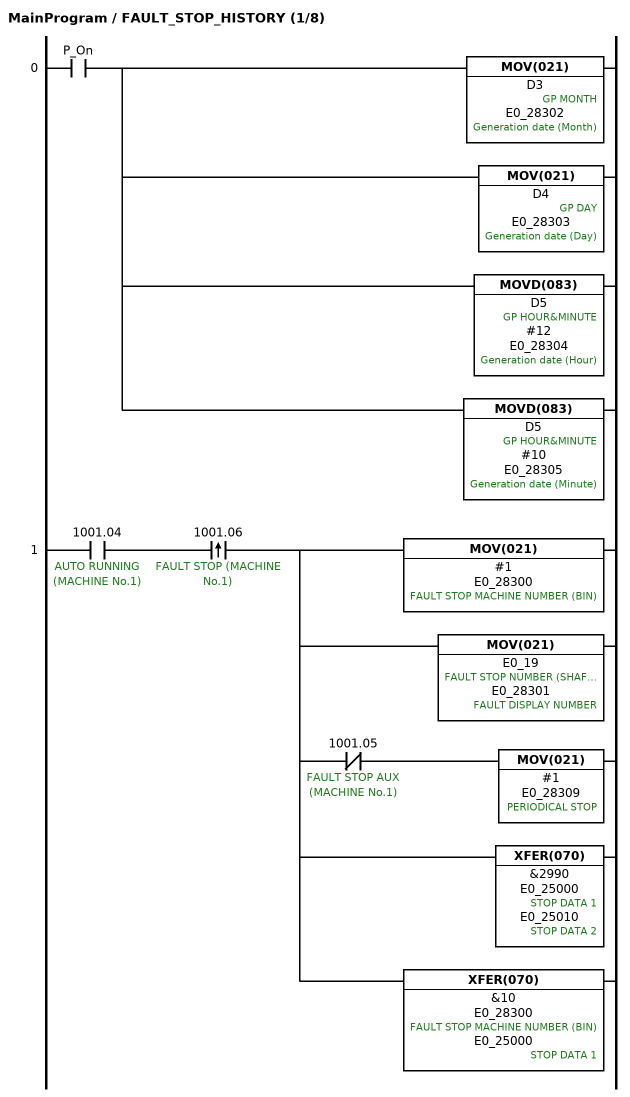
; [picture p168: MainProgram / FAULT_STOP_HISTORY, rungs 0-1]
; rung 0
LD P_On
MOV(021) D3 E0_28302  ; GP MONTH, Generation date (Month)
MOV(021) D4 E0_28303  ; GP DAY, Generation date (Day)
MOVD(083) D5 #12 E0_28304  ; GP HOUR&MINUTE, Generation date (Hour)
MOVD(083) D5 #10 E0_28305  ; GP HOUR&MINUTE, Generation date (Minute)
; rung 1
LD 1001.04  ; AUTO RUNNING (MACHINE No.1)
@AND 1001.06  ; FAULT STOP (MACHINE No.1)
OUT TR0
MOV(021) #1 E0_28300  ; FAULT STOP MACHINE NUMBER (BIN)
MOV(021) E0_19 E0_28301  ; FAULT STOP NUMBER (SHAFT PRESS-FITTING), FAULT DISPLAY NUMBER
ANDNOT 1001.05  ; FAULT STOP AUX (MACHINE No.1)
MOV(021) #1 E0_28309  ; PERIODICAL STOP
LD TR0
XFER(070) &2990 E0_25000 E0_25010  ; STOP DATA 1, STOP DATA 2
XFER(070) &10 E0_28300 E0_25000  ; FAULT STOP MACHINE NUMBER (BIN), STOP DATA 1

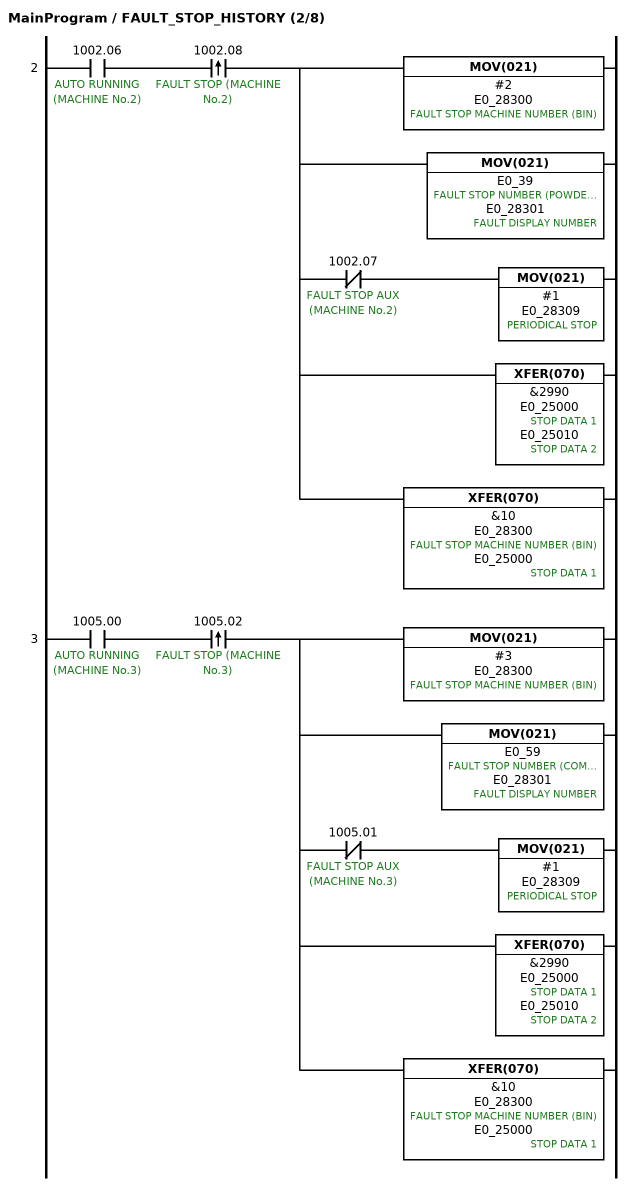
; rung 2
LD 1002.06  ; AUTO RUNNING (MACHINE No.2)
@AND 1002.08  ; FAULT STOP (MACHINE No.2)
OUT TR0
MOV(021) #2 E0_28300  ; FAULT STOP MACHINE NUMBER (BIN)
MOV(021) E0_39 E0_28301  ; FAULT STOP NUMBER (POWDER COATING), FAULT DISPLAY NUMBER
ANDNOT 1002.07  ; FAULT STOP AUX (MACHINE No.2)
MOV(021) #1 E0_28309  ; PERIODICAL STOP
LD TR0
XFER(070) &2990 E0_25000 E0_25010  ; STOP DATA 1, STOP DATA 2
XFER(070) &10 E0_28300 E0_25000  ; FAULT STOP MACHINE NUMBER (BIN), STOP DATA 1
; rung 3
LD 1005.00  ; AUTO RUNNING (MACHINE No.3)
@AND 1005.02  ; FAULT STOP (MACHINE No.3)
OUT TR0
MOV(021) #3 E0_28300  ; FAULT STOP MACHINE NUMBER (BIN)
MOV(021) E0_59 E0_28301  ; FAULT STOP NUMBER (COMM PRESS-FITTING), FAULT DISPLAY NUMBER
ANDNOT 1005.01  ; FAULT STOP AUX (MACHINE No.3)
MOV(021) #1 E0_28309  ; PERIODICAL STOP
LD TR0
XFER(070) &2990 E0_25000 E0_25010  ; STOP DATA 1, STOP DATA 2
XFER(070) &10 E0_28300 E0_25000  ; FAULT STOP MACHINE NUMBER (BIN), STOP DATA 1

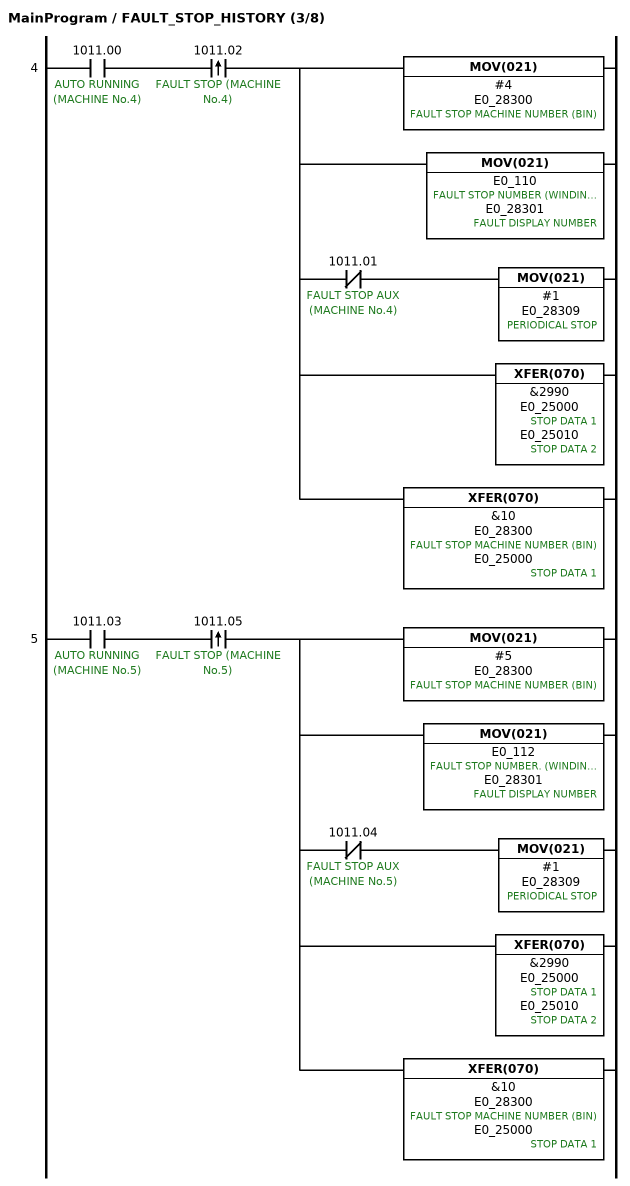
; rung 4
LD 1011.00  ; AUTO RUNNING (MACHINE No.4)
@AND 1011.02  ; FAULT STOP (MACHINE No.4)
OUT TR0
MOV(021) #4 E0_28300  ; FAULT STOP MACHINE NUMBER (BIN)
MOV(021) E0_110 E0_28301  ; FAULT STOP NUMBER (WINDING No.1), FAULT DISPLAY NUMBER
ANDNOT 1011.01  ; FAULT STOP AUX (MACHINE No.4)
MOV(021) #1 E0_28309  ; PERIODICAL STOP
LD TR0
XFER(070) &2990 E0_25000 E0_25010  ; STOP DATA 1, STOP DATA 2
XFER(070) &10 E0_28300 E0_25000  ; FAULT STOP MACHINE NUMBER (BIN), STOP DATA 1
; rung 5
LD 1011.03  ; AUTO RUNNING (MACHINE No.5)
@AND 1011.05  ; FAULT STOP (MACHINE No.5)
OUT TR0
MOV(021) #5 E0_28300  ; FAULT STOP MACHINE NUMBER (BIN)
MOV(021) E0_112 E0_28301  ; FAULT STOP NUMBER. (WINDING No.2), FAULT DISPLAY NUMBER
ANDNOT 1011.04  ; FAULT STOP AUX (MACHINE No.5)
MOV(021) #1 E0_28309  ; PERIODICAL STOP
LD TR0
XFER(070) &2990 E0_25000 E0_25010  ; STOP DATA 1, STOP DATA 2
XFER(070) &10 E0_28300 E0_25000  ; FAULT STOP MACHINE NUMBER (BIN), STOP DATA 1

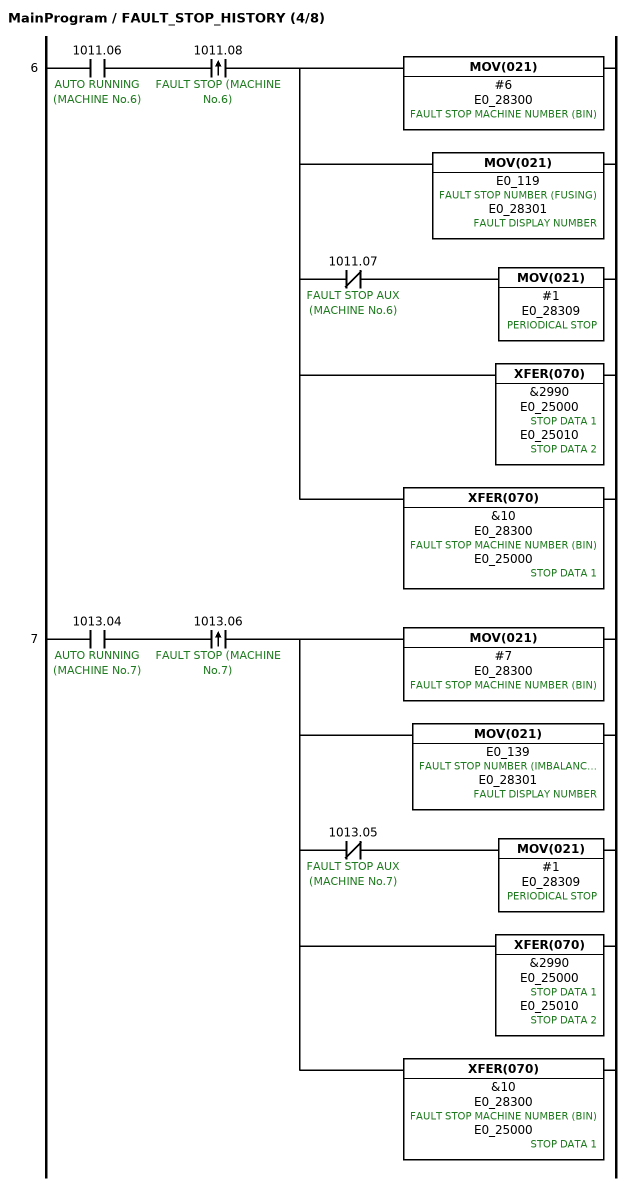
; rung 6
LD 1011.06  ; AUTO RUNNING (MACHINE No.6)
@AND 1011.08  ; FAULT STOP (MACHINE No.6)
OUT TR0
MOV(021) #6 E0_28300  ; FAULT STOP MACHINE NUMBER (BIN)
MOV(021) E0_119 E0_28301  ; FAULT STOP NUMBER (FUSING), FAULT DISPLAY NUMBER
ANDNOT 1011.07  ; FAULT STOP AUX (MACHINE No.6)
MOV(021) #1 E0_28309  ; PERIODICAL STOP
LD TR0
XFER(070) &2990 E0_25000 E0_25010  ; STOP DATA 1, STOP DATA 2
XFER(070) &10 E0_28300 E0_25000  ; FAULT STOP MACHINE NUMBER (BIN), STOP DATA 1
; rung 7
LD 1013.04  ; AUTO RUNNING (MACHINE No.7)
@AND 1013.06  ; FAULT STOP (MACHINE No.7)
OUT TR0
MOV(021) #7 E0_28300  ; FAULT STOP MACHINE NUMBER (BIN)
MOV(021) E0_139 E0_28301  ; FAULT STOP NUMBER (IMBALANCE CORRECTING), FAULT DISPLAY NUMBER
ANDNOT 1013.05  ; FAULT STOP AUX (MACHINE No.7)
MOV(021) #1 E0_28309  ; PERIODICAL STOP
LD TR0
XFER(070) &2990 E0_25000 E0_25010  ; STOP DATA 1, STOP DATA 2
XFER(070) &10 E0_28300 E0_25000  ; FAULT STOP MACHINE NUMBER (BIN), STOP DATA 1

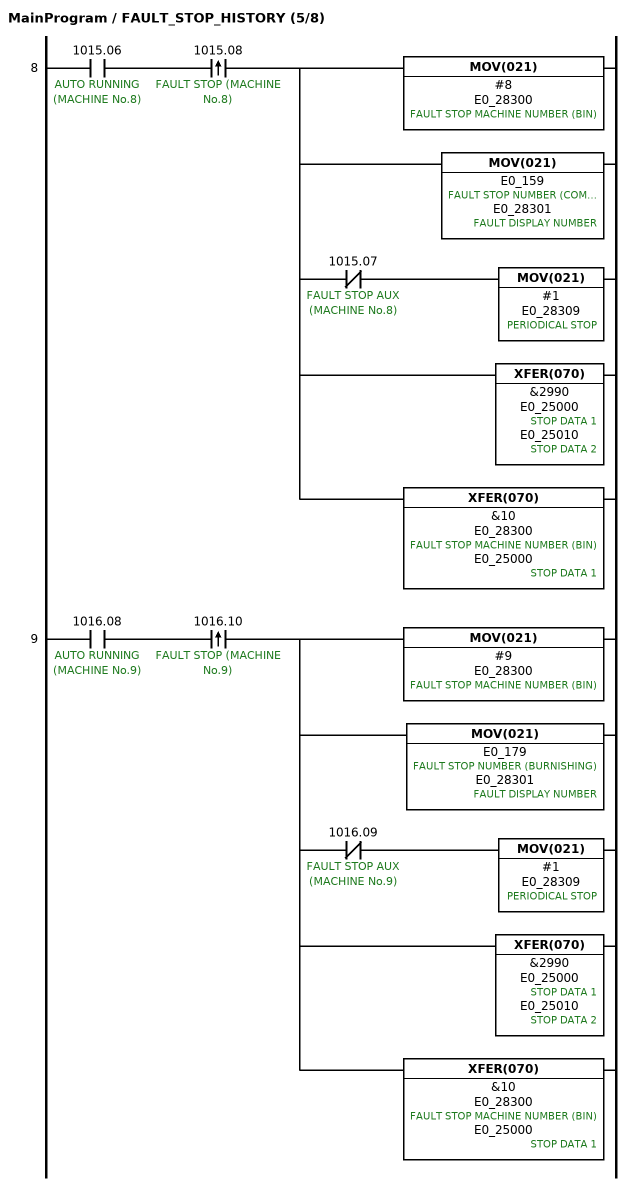
; rung 8
LD 1015.06  ; AUTO RUNNING (MACHINE No.8)
@AND 1015.08  ; FAULT STOP (MACHINE No.8)
OUT TR0
MOV(021) #8 E0_28300  ; FAULT STOP MACHINE NUMBER (BIN)
MOV(021) E0_159 E0_28301  ; FAULT STOP NUMBER (COMM TURNING), FAULT DISPLAY NUMBER
ANDNOT 1015.07  ; FAULT STOP AUX (MACHINE No.8)
MOV(021) #1 E0_28309  ; PERIODICAL STOP
LD TR0
XFER(070) &2990 E0_25000 E0_25010  ; STOP DATA 1, STOP DATA 2
XFER(070) &10 E0_28300 E0_25000  ; FAULT STOP MACHINE NUMBER (BIN), STOP DATA 1
; rung 9
LD 1016.08  ; AUTO RUNNING (MACHINE No.9)
@AND 1016.10  ; FAULT STOP (MACHINE No.9)
OUT TR0
MOV(021) #9 E0_28300  ; FAULT STOP MACHINE NUMBER (BIN)
MOV(021) E0_179 E0_28301  ; FAULT STOP NUMBER (BURNISHING), FAULT DISPLAY NUMBER
ANDNOT 1016.09  ; FAULT STOP AUX (MACHINE No.9)
MOV(021) #1 E0_28309  ; PERIODICAL STOP
LD TR0
XFER(070) &2990 E0_25000 E0_25010  ; STOP DATA 1, STOP DATA 2
XFER(070) &10 E0_28300 E0_25000  ; FAULT STOP MACHINE NUMBER (BIN), STOP DATA 1

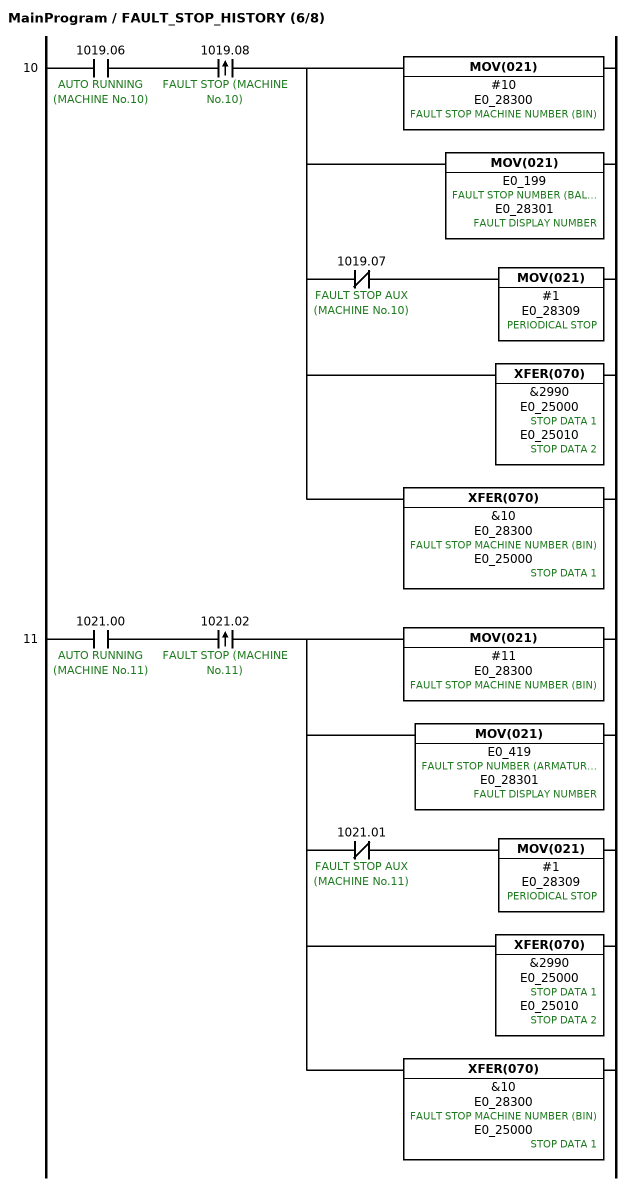
; rung 10
LD 1019.06  ; AUTO RUNNING (MACHINE No.10)
@AND 1019.08  ; FAULT STOP (MACHINE No.10)
OUT TR0
MOV(021) #10 E0_28300  ; FAULT STOP MACHINE NUMBER (BIN)
MOV(021) E0_199 E0_28301  ; FAULT STOP NUMBER (BALL STACKING), FAULT DISPLAY NUMBER
ANDNOT 1019.07  ; FAULT STOP AUX (MACHINE No.10)
MOV(021) #1 E0_28309  ; PERIODICAL STOP
LD TR0
XFER(070) &2990 E0_25000 E0_25010  ; STOP DATA 1, STOP DATA 2
XFER(070) &10 E0_28300 E0_25000  ; FAULT STOP MACHINE NUMBER (BIN), STOP DATA 1
; rung 11
LD 1021.00  ; AUTO RUNNING (MACHINE No.11)
@AND 1021.02  ; FAULT STOP (MACHINE No.11)
OUT TR0
MOV(021) #11 E0_28300  ; FAULT STOP MACHINE NUMBER (BIN)
MOV(021) E0_419 E0_28301  ; FAULT STOP NUMBER (ARMATURE TESTER), FAULT DISPLAY NUMBER
ANDNOT 1021.01  ; FAULT STOP AUX (MACHINE No.11)
MOV(021) #1 E0_28309  ; PERIODICAL STOP
LD TR0
XFER(070) &2990 E0_25000 E0_25010  ; STOP DATA 1, STOP DATA 2
XFER(070) &10 E0_28300 E0_25000  ; FAULT STOP MACHINE NUMBER (BIN), STOP DATA 1

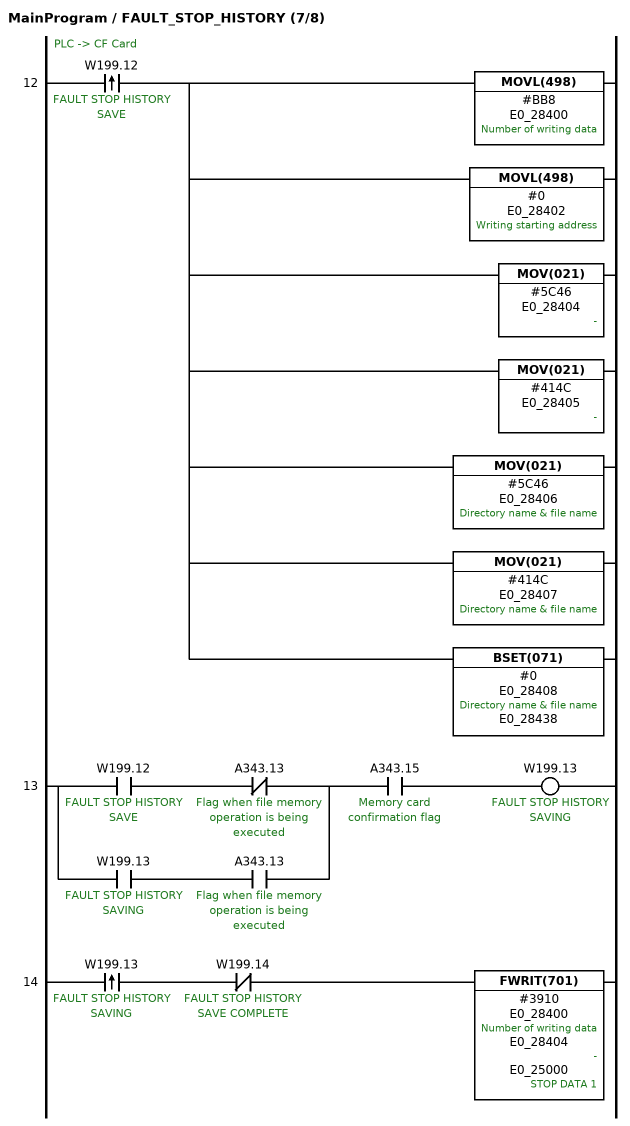
; rung 12: PLC -> CF Card
@LD W199.12  ; FAULT STOP HISTORY SAVE
MOVL(498) #BB8 E0_28400  ; Number of writing data  // Number of data (BB8HEX (3000BCD))
MOVL(498) #0 E0_28402  ; Writing starting address
MOV(021) #5C46 E0_28404  ; -  // 'Directory name"FAL"'
MOV(021) #414C E0_28405  ; -
MOV(021) #5C46 E0_28406  ; Directory name & file name  // 'File name"FAL"'
MOV(021) #414C E0_28407  ; Directory name & file name
BSET(071) #0 E0_28408 E0_28438  ; Directory name & file name
; rung 13
LD W199.12  ; FAULT STOP HISTORY SAVE
ANDNOT A343.13  ; Flag when file memory operation is being executed
LD W199.13  ; FAULT STOP HISTORY SAVING
AND A343.13  ; Flag when file memory operation is being executed
ORLD
AND A343.15  ; Memory card confirmation flag
OUT W199.13  ; FAULT STOP HISTORY SAVING
; rung 14
@LD W199.13  ; FAULT STOP HISTORY SAVING
ANDNOT W199.14  ; FAULT STOP HISTORY SAVE COMPLETE
FWRIT(701) #3910 E0_28400 E0_28404 E0_25000  ; Number of writing data, -, STOP DATA 1

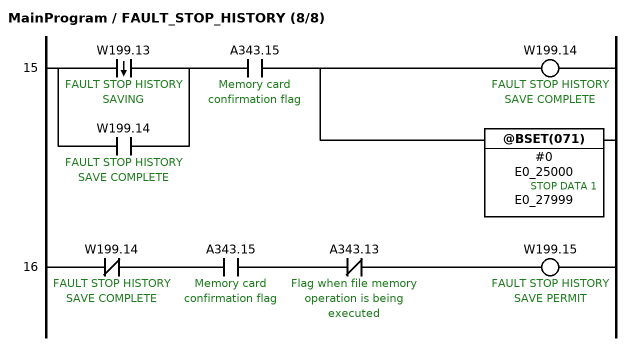
; rung 15
%LD W199.13  ; FAULT STOP HISTORY SAVING
OR W199.14  ; FAULT STOP HISTORY SAVE COMPLETE
AND A343.15  ; Memory card confirmation flag
OUT W199.14  ; FAULT STOP HISTORY SAVE COMPLETE
@BSET(071) #0 E0_25000 E0_27999  ; STOP DATA 1
; rung 16
LDNOT W199.14  ; FAULT STOP HISTORY SAVE COMPLETE
AND A343.15  ; Memory card confirmation flag
ANDNOT A343.13  ; Flag when file memory operation is being executed
OUT W199.15  ; FAULT STOP HISTORY SAVE PERMIT

### Section SHORT_STOP_HISTORY

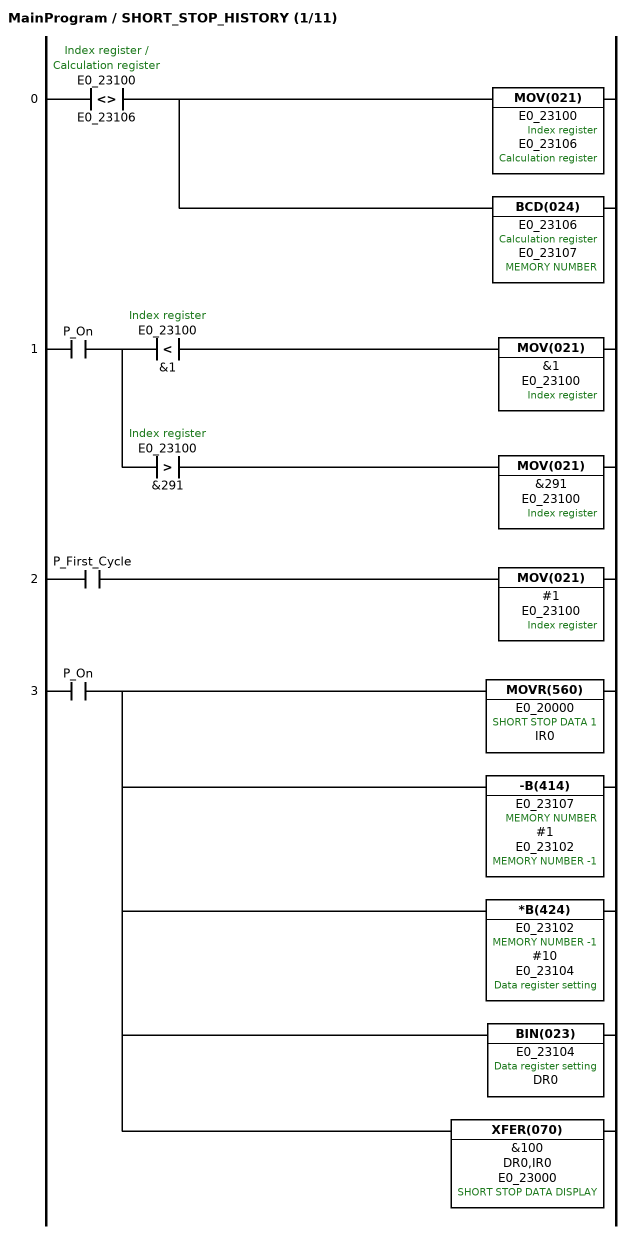
; rung 0
LD<>(305) E0_23100 E0_23106  ; Index register, Calculation register
MOV(021) E0_23100 E0_23106  ; Index register, Calculation register
BCD(024) E0_23106 E0_23107  ; Calculation register, MEMORY NUMBER
; rung 1
LD P_On
OUT TR0
AND<(310) E0_23100 &1  ; Index register
MOV(021) &1 E0_23100  ; Index register
LD TR0
AND>(320) E0_23100 &291  ; Index register
MOV(021) &291 E0_23100  ; Index register
; rung 2
LD P_First_Cycle
MOV(021) #1 E0_23100  ; Index register
; rung 3
LD P_On
MOVR(560) E0_20000 IR0  ; SHORT STOP DATA 1
-B(414) E0_23107 #1 E0_23102  ; MEMORY NUMBER, MEMORY NUMBER -1
*B(424) E0_23102 #10 E0_23104  ; MEMORY NUMBER -1, Data register setting
BIN(023) E0_23104 DR0  ; Data register setting
XFER(070) &100 DR0,IR0 E0_23000  ; SHORT STOP DATA DISPLAY

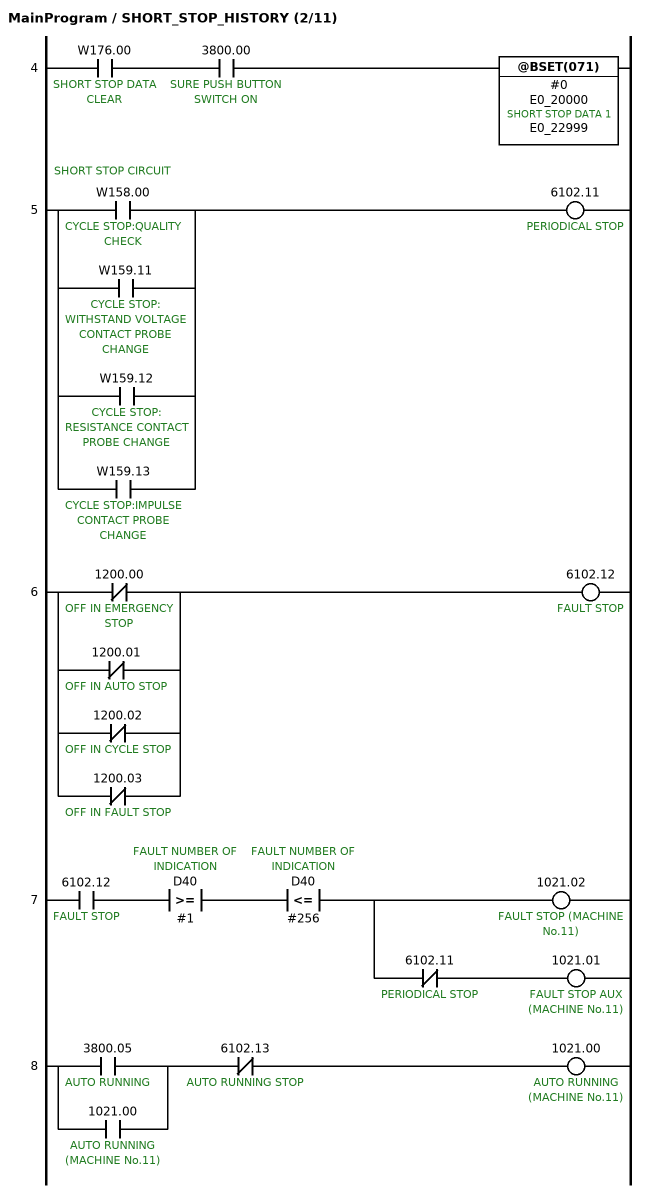
; rung 4
LD W176.00  ; SHORT STOP DATA CLEAR
AND 3800.00  ; SURE PUSH BUTTON SWITCH ON
@BSET(071) #0 E0_20000 E0_22999  ; SHORT STOP DATA 1
; rung 5: SHORT STOP CIRCUIT
LD W158.00  ; CYCLE STOP:QUALITY CHECK
OR W159.11  ; CYCLE STOP:WITHSTAND VOLTAGE CONTACT PROBE CHANGE
OR W159.12  ; CYCLE STOP:RESISTANCE CONTACT PROBE CHANGE
OR W159.13  ; CYCLE STOP:IMPULSE CONTACT PROBE CHANGE
OUT 6102.11  ; PERIODICAL STOP
; rung 6
LDNOT 1200.00  ; OFF IN EMERGENCY STOP
ORNOT 1200.01  ; OFF IN AUTO STOP
ORNOT 1200.02  ; OFF IN CYCLE STOP
ORNOT 1200.03  ; OFF IN FAULT STOP
OUT 6102.12  ; FAULT STOP
; rung 7
LD 6102.12  ; FAULT STOP
AND>=(325) D40 #1  ; FAULT NUMBER OF INDICATION
AND<=(315) D40 #256  ; FAULT NUMBER OF INDICATION
OUT 1021.02  ; FAULT STOP (MACHINE No.11)
ANDNOT 6102.11  ; PERIODICAL STOP
OUT 1021.01  ; FAULT STOP AUX (MACHINE No.11)
; rung 8
LD 3800.05  ; AUTO RUNNING
OR 1021.00  ; AUTO RUNNING (MACHINE No.11)
ANDNOT 6102.13  ; AUTO RUNNING STOP
OUT 1021.00  ; AUTO RUNNING (MACHINE No.11)

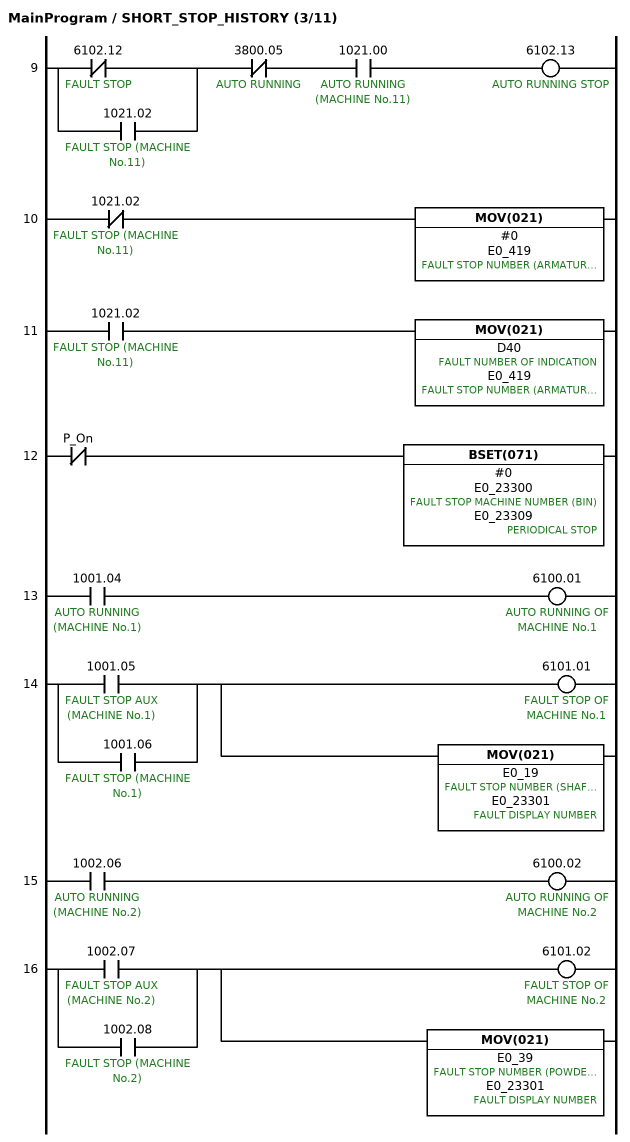
; rung 9
LDNOT 6102.12  ; FAULT STOP
OR 1021.02  ; FAULT STOP (MACHINE No.11)
ANDNOT 3800.05  ; AUTO RUNNING
AND 1021.00  ; AUTO RUNNING (MACHINE No.11)
OUT 6102.13  ; AUTO RUNNING STOP
; rung 10
LDNOT 1021.02  ; FAULT STOP (MACHINE No.11)
MOV(021) #0 E0_419  ; FAULT STOP NUMBER (ARMATURE TESTER)
; rung 11
LD 1021.02  ; FAULT STOP (MACHINE No.11)
MOV(021) D40 E0_419  ; FAULT NUMBER OF INDICATION, FAULT STOP NUMBER (ARMATURE TESTER)
; rung 12
LDNOT P_On
BSET(071) #0 E0_23300 E0_23309  ; FAULT STOP MACHINE NUMBER (BIN), PERIODICAL STOP
; rung 13
LD 1001.04  ; AUTO RUNNING (MACHINE No.1)
OUT 6100.01  ; AUTO RUNNING OF MACHINE No.1
; rung 14
LD 1001.05  ; FAULT STOP AUX (MACHINE No.1)
OR 1001.06  ; FAULT STOP (MACHINE No.1)
OUT 6101.01  ; FAULT STOP OF MACHINE No.1
MOV(021) E0_19 E0_23301  ; FAULT STOP NUMBER (SHAFT PRESS-FITTING), FAULT DISPLAY NUMBER
; rung 15
LD 1002.06  ; AUTO RUNNING (MACHINE No.2)
OUT 6100.02  ; AUTO RUNNING OF MACHINE No.2
; rung 16
LD 1002.07  ; FAULT STOP AUX (MACHINE No.2)
OR 1002.08  ; FAULT STOP (MACHINE No.2)
OUT 6101.02  ; FAULT STOP OF MACHINE No.2
MOV(021) E0_39 E0_23301  ; FAULT STOP NUMBER (POWDER COATING), FAULT DISPLAY NUMBER

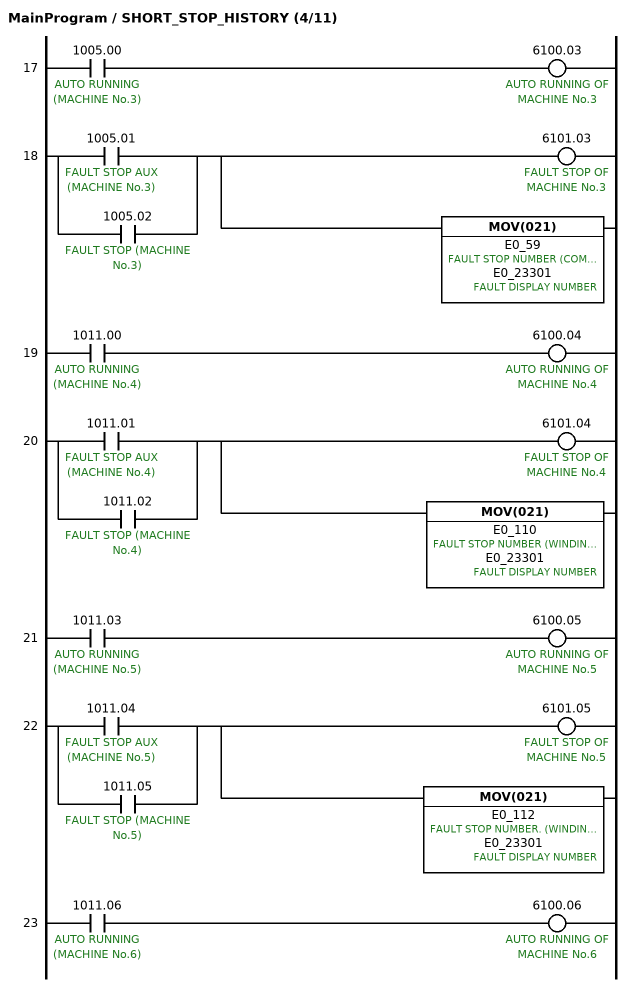
; rung 17
LD 1005.00  ; AUTO RUNNING (MACHINE No.3)
OUT 6100.03  ; AUTO RUNNING OF MACHINE No.3
; rung 18
LD 1005.01  ; FAULT STOP AUX (MACHINE No.3)
OR 1005.02  ; FAULT STOP (MACHINE No.3)
OUT 6101.03  ; FAULT STOP OF MACHINE No.3
MOV(021) E0_59 E0_23301  ; FAULT STOP NUMBER (COMM PRESS-FITTING), FAULT DISPLAY NUMBER
; rung 19
LD 1011.00  ; AUTO RUNNING (MACHINE No.4)
OUT 6100.04  ; AUTO RUNNING OF MACHINE No.4
; rung 20
LD 1011.01  ; FAULT STOP AUX (MACHINE No.4)
OR 1011.02  ; FAULT STOP (MACHINE No.4)
OUT 6101.04  ; FAULT STOP OF MACHINE No.4
MOV(021) E0_110 E0_23301  ; FAULT STOP NUMBER (WINDING No.1), FAULT DISPLAY NUMBER
; rung 21
LD 1011.03  ; AUTO RUNNING (MACHINE No.5)
OUT 6100.05  ; AUTO RUNNING OF MACHINE No.5
; rung 22
LD 1011.04  ; FAULT STOP AUX (MACHINE No.5)
OR 1011.05  ; FAULT STOP (MACHINE No.5)
OUT 6101.05  ; FAULT STOP OF MACHINE No.5
MOV(021) E0_112 E0_23301  ; FAULT STOP NUMBER. (WINDING No.2), FAULT DISPLAY NUMBER
; rung 23
LD 1011.06  ; AUTO RUNNING (MACHINE No.6)
OUT 6100.06  ; AUTO RUNNING OF MACHINE No.6

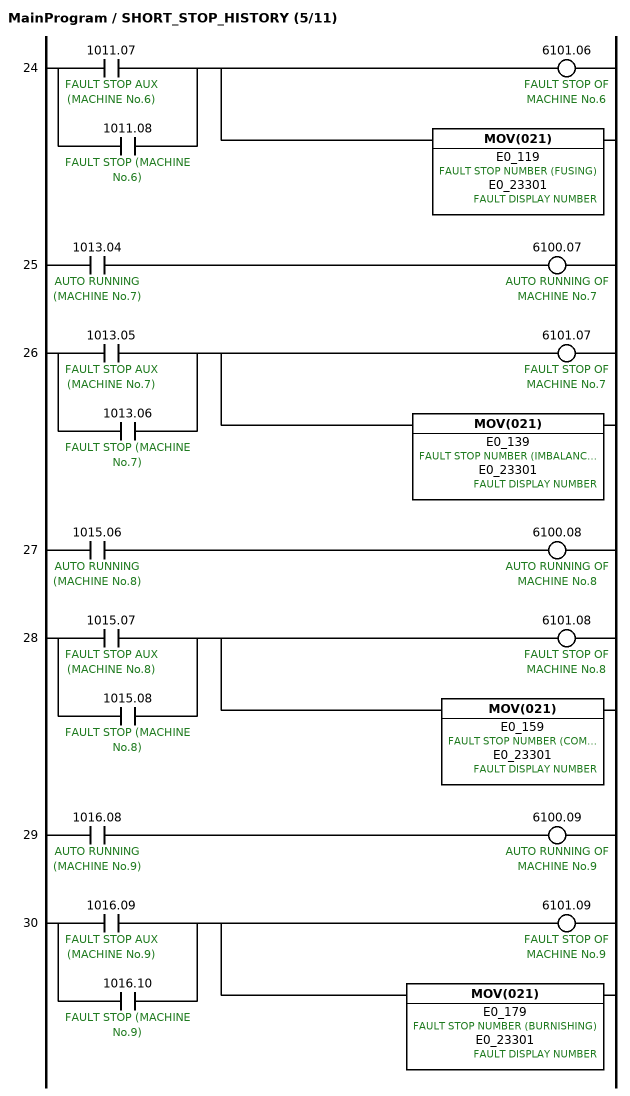
; rung 24
LD 1011.07  ; FAULT STOP AUX (MACHINE No.6)
OR 1011.08  ; FAULT STOP (MACHINE No.6)
OUT 6101.06  ; FAULT STOP OF MACHINE No.6
MOV(021) E0_119 E0_23301  ; FAULT STOP NUMBER (FUSING), FAULT DISPLAY NUMBER
; rung 25
LD 1013.04  ; AUTO RUNNING (MACHINE No.7)
OUT 6100.07  ; AUTO RUNNING OF MACHINE No.7
; rung 26
LD 1013.05  ; FAULT STOP AUX (MACHINE No.7)
OR 1013.06  ; FAULT STOP (MACHINE No.7)
OUT 6101.07  ; FAULT STOP OF MACHINE No.7
MOV(021) E0_139 E0_23301  ; FAULT STOP NUMBER (IMBALANCE CORRECTING), FAULT DISPLAY NUMBER
; rung 27
LD 1015.06  ; AUTO RUNNING (MACHINE No.8)
OUT 6100.08  ; AUTO RUNNING OF MACHINE No.8
; rung 28
LD 1015.07  ; FAULT STOP AUX (MACHINE No.8)
OR 1015.08  ; FAULT STOP (MACHINE No.8)
OUT 6101.08  ; FAULT STOP OF MACHINE No.8
MOV(021) E0_159 E0_23301  ; FAULT STOP NUMBER (COMM TURNING), FAULT DISPLAY NUMBER
; rung 29
LD 1016.08  ; AUTO RUNNING (MACHINE No.9)
OUT 6100.09  ; AUTO RUNNING OF MACHINE No.9
; rung 30
LD 1016.09  ; FAULT STOP AUX (MACHINE No.9)
OR 1016.10  ; FAULT STOP (MACHINE No.9)
OUT 6101.09  ; FAULT STOP OF MACHINE No.9
MOV(021) E0_179 E0_23301  ; FAULT STOP NUMBER (BURNISHING), FAULT DISPLAY NUMBER

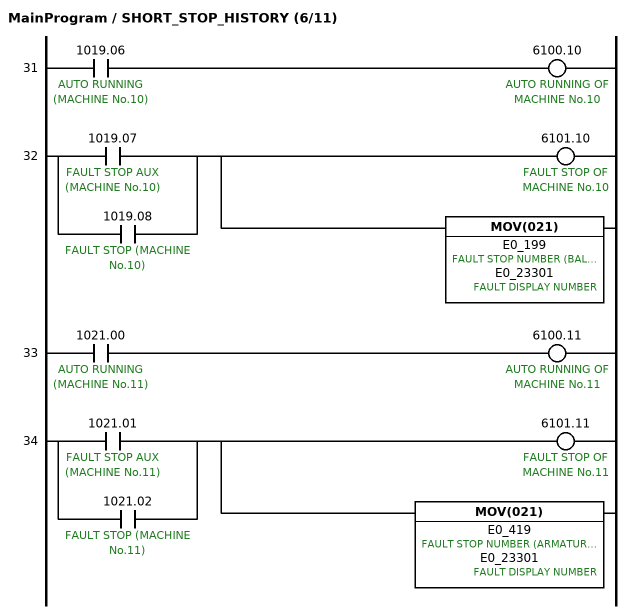
; rung 31
LD 1019.06  ; AUTO RUNNING (MACHINE No.10)
OUT 6100.10  ; AUTO RUNNING OF MACHINE No.10
; rung 32
LD 1019.07  ; FAULT STOP AUX (MACHINE No.10)
OR 1019.08  ; FAULT STOP (MACHINE No.10)
OUT 6101.10  ; FAULT STOP OF MACHINE No.10
MOV(021) E0_199 E0_23301  ; FAULT STOP NUMBER (BALL STACKING), FAULT DISPLAY NUMBER
; rung 33
LD 1021.00  ; AUTO RUNNING (MACHINE No.11)
OUT 6100.11  ; AUTO RUNNING OF MACHINE No.11
; rung 34
LD 1021.01  ; FAULT STOP AUX (MACHINE No.11)
OR 1021.02  ; FAULT STOP (MACHINE No.11)
OUT 6101.11  ; FAULT STOP OF MACHINE No.11
MOV(021) E0_419 E0_23301  ; FAULT STOP NUMBER (ARMATURE TESTER), FAULT DISPLAY NUMBER

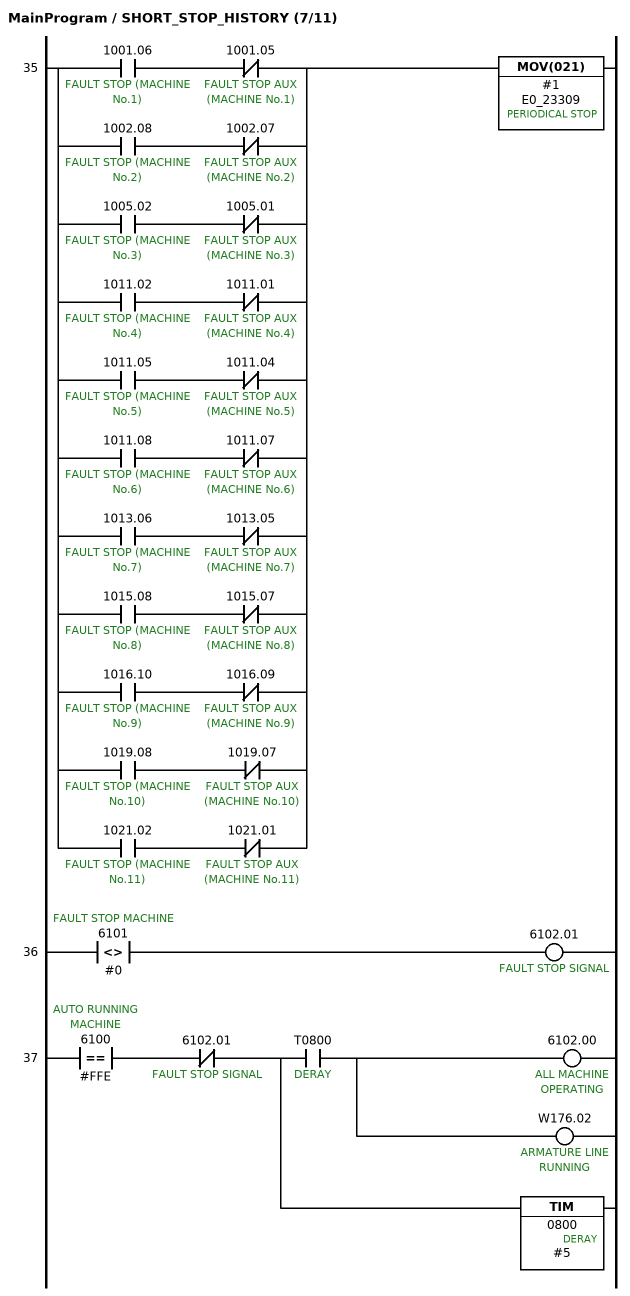
; rung 35
LD 1001.06  ; FAULT STOP (MACHINE No.1)
ANDNOT 1001.05  ; FAULT STOP AUX (MACHINE No.1)
LD 1002.08  ; FAULT STOP (MACHINE No.2)
ANDNOT 1002.07  ; FAULT STOP AUX (MACHINE No.2)
ORLD
LD 1005.02  ; FAULT STOP (MACHINE No.3)
ANDNOT 1005.01  ; FAULT STOP AUX (MACHINE No.3)
ORLD
LD 1011.02  ; FAULT STOP (MACHINE No.4)
ANDNOT 1011.01  ; FAULT STOP AUX (MACHINE No.4)
ORLD
LD 1011.05  ; FAULT STOP (MACHINE No.5)
ANDNOT 1011.04  ; FAULT STOP AUX (MACHINE No.5)
ORLD
LD 1011.08  ; FAULT STOP (MACHINE No.6)
ANDNOT 1011.07  ; FAULT STOP AUX (MACHINE No.6)
ORLD
LD 1013.06  ; FAULT STOP (MACHINE No.7)
ANDNOT 1013.05  ; FAULT STOP AUX (MACHINE No.7)
ORLD
LD 1015.08  ; FAULT STOP (MACHINE No.8)
ANDNOT 1015.07  ; FAULT STOP AUX (MACHINE No.8)
ORLD
LD 1016.10  ; FAULT STOP (MACHINE No.9)
ANDNOT 1016.09  ; FAULT STOP AUX (MACHINE No.9)
ORLD
LD 1019.08  ; FAULT STOP (MACHINE No.10)
ANDNOT 1019.07  ; FAULT STOP AUX (MACHINE No.10)
ORLD
LD 1021.02  ; FAULT STOP (MACHINE No.11)
ANDNOT 1021.01  ; FAULT STOP AUX (MACHINE No.11)
ORLD
MOV(021) #1 E0_23309  ; PERIODICAL STOP
; rung 36
LD<>(305) 6101 #0  ; FAULT STOP MACHINE
OUT 6102.01  ; FAULT STOP SIGNAL
; rung 37
LD=(300) 6100 #FFE  ; AUTO RUNNING MACHINE
ANDNOT 6102.01  ; FAULT STOP SIGNAL
OUT TR0
AND T0800  ; DERAY
OUT 6102.00  ; ALL MACHINE OPERATING
OUT W176.02  ; ARMATURE LINE RUNNING
LD TR0
TIM 0800 #5  ; DERAY

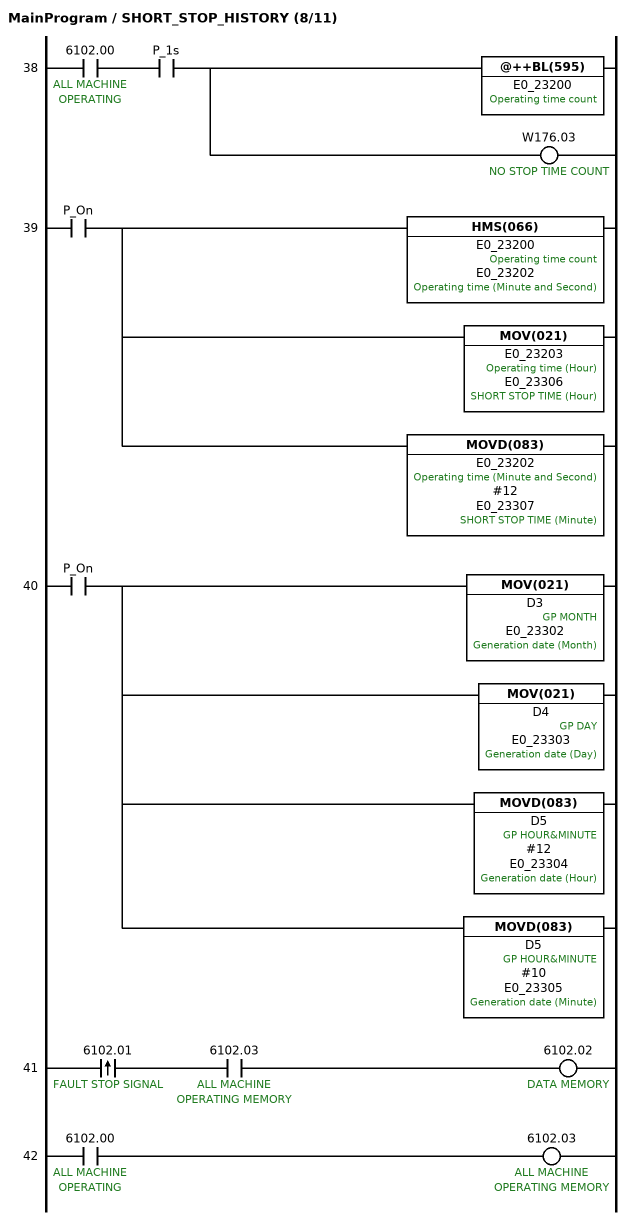
; rung 38
LD 6102.00  ; ALL MACHINE OPERATING
AND P_1s
@++BL(595) E0_23200  ; Operating time count
OUT W176.03  ; NO STOP TIME COUNT
; rung 39
LD P_On
HMS(066) E0_23200 E0_23202  ; Operating time count, Operating time (Minute and Second)
MOV(021) E0_23203 E0_23306  ; Operating time (Hour), SHORT STOP TIME (Hour)
MOVD(083) E0_23202 #12 E0_23307  ; Operating time (Minute and Second), SHORT STOP TIME (Minute)
; rung 40
LD P_On
MOV(021) D3 E0_23302  ; GP MONTH, Generation date (Month)
MOV(021) D4 E0_23303  ; GP DAY, Generation date (Day)
MOVD(083) D5 #12 E0_23304  ; GP HOUR&MINUTE, Generation date (Hour)
MOVD(083) D5 #10 E0_23305  ; GP HOUR&MINUTE, Generation date (Minute)
; rung 41
@LD 6102.01  ; FAULT STOP SIGNAL
AND 6102.03  ; ALL MACHINE OPERATING MEMORY
OUT 6102.02  ; DATA MEMORY
; rung 42
LD 6102.00  ; ALL MACHINE OPERATING
OUT 6102.03  ; ALL MACHINE OPERATING MEMORY

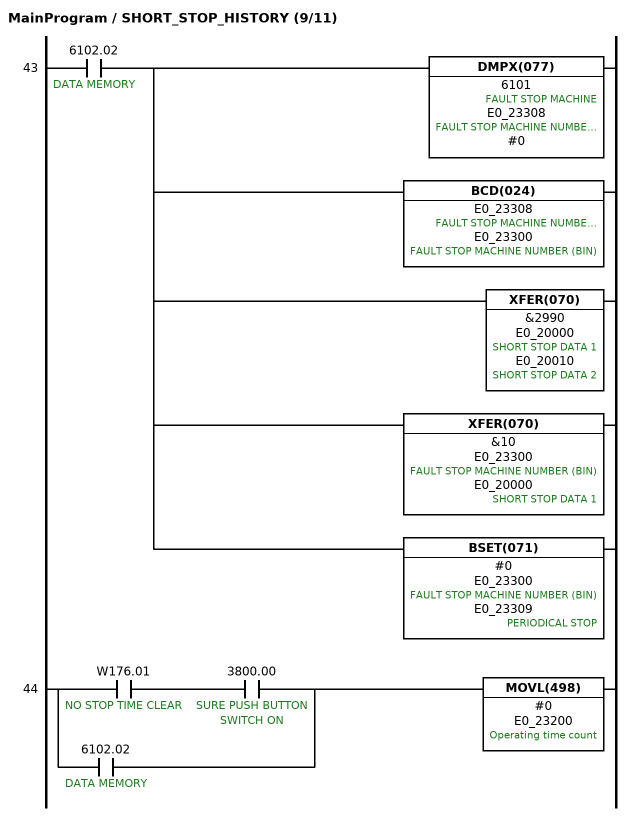
; rung 43
LD 6102.02  ; DATA MEMORY
DMPX(077) 6101 E0_23308 #0  ; FAULT STOP MACHINE, FAULT STOP MACHINE NUMBER (BCD)
BCD(024) E0_23308 E0_23300  ; FAULT STOP MACHINE NUMBER (BCD), FAULT STOP MACHINE NUMBER (BIN)
XFER(070) &2990 E0_20000 E0_20010  ; SHORT STOP DATA 1, SHORT STOP DATA 2
XFER(070) &10 E0_23300 E0_20000  ; FAULT STOP MACHINE NUMBER (BIN), SHORT STOP DATA 1
BSET(071) #0 E0_23300 E0_23309  ; FAULT STOP MACHINE NUMBER (BIN), PERIODICAL STOP
; rung 44
LD W176.01  ; NO STOP TIME CLEAR
AND 3800.00  ; SURE PUSH BUTTON SWITCH ON
OR 6102.02  ; DATA MEMORY
MOVL(498) #0 E0_23200  ; Operating time count

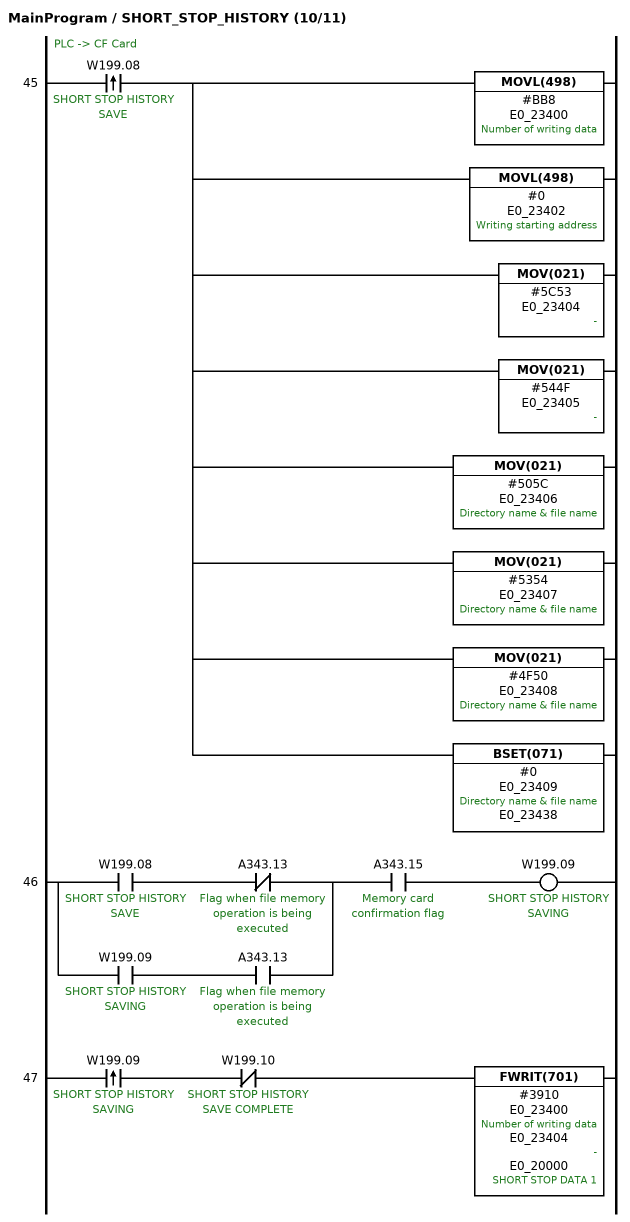
; rung 45: PLC -> CF Card
@LD W199.08  ; SHORT STOP HISTORY SAVE
MOVL(498) #BB8 E0_23400  ; Number of writing data  // Number of data (BB8HEX (3000BCD))
MOVL(498) #0 E0_23402  ; Writing starting address
MOV(021) #5C53 E0_23404  ; -  // 'Directory name"STOP"'
MOV(021) #544F E0_23405  ; -
MOV(021) #505C E0_23406  ; Directory name & file name
MOV(021) #5354 E0_23407  ; Directory name & file name  // 'File name"STOP"'
MOV(021) #4F50 E0_23408  ; Directory name & file name
BSET(071) #0 E0_23409 E0_23438  ; Directory name & file name
; rung 46
LD W199.08  ; SHORT STOP HISTORY SAVE
ANDNOT A343.13  ; Flag when file memory operation is being executed
LD W199.09  ; SHORT STOP HISTORY SAVING
AND A343.13  ; Flag when file memory operation is being executed
ORLD
AND A343.15  ; Memory card confirmation flag
OUT W199.09  ; SHORT STOP HISTORY SAVING
; rung 47
@LD W199.09  ; SHORT STOP HISTORY SAVING
ANDNOT W199.10  ; SHORT STOP HISTORY SAVE COMPLETE
FWRIT(701) #3910 E0_23400 E0_23404 E0_20000  ; Number of writing data, -, SHORT STOP DATA 1

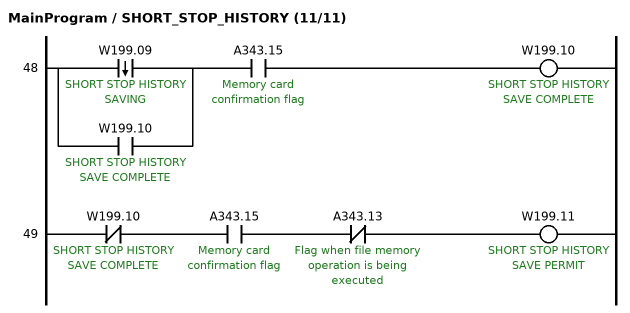
; rung 48
%LD W199.09  ; SHORT STOP HISTORY SAVING
OR W199.10  ; SHORT STOP HISTORY SAVE COMPLETE
AND A343.15  ; Memory card confirmation flag
OUT W199.10  ; SHORT STOP HISTORY SAVE COMPLETE
; rung 49
LDNOT W199.10  ; SHORT STOP HISTORY SAVE COMPLETE
AND A343.15  ; Memory card confirmation flag
ANDNOT A343.13  ; Flag when file memory operation is being executed
OUT W199.11  ; SHORT STOP HISTORY SAVE PERMIT

### Section UNLOADING_LANE_SET_UP

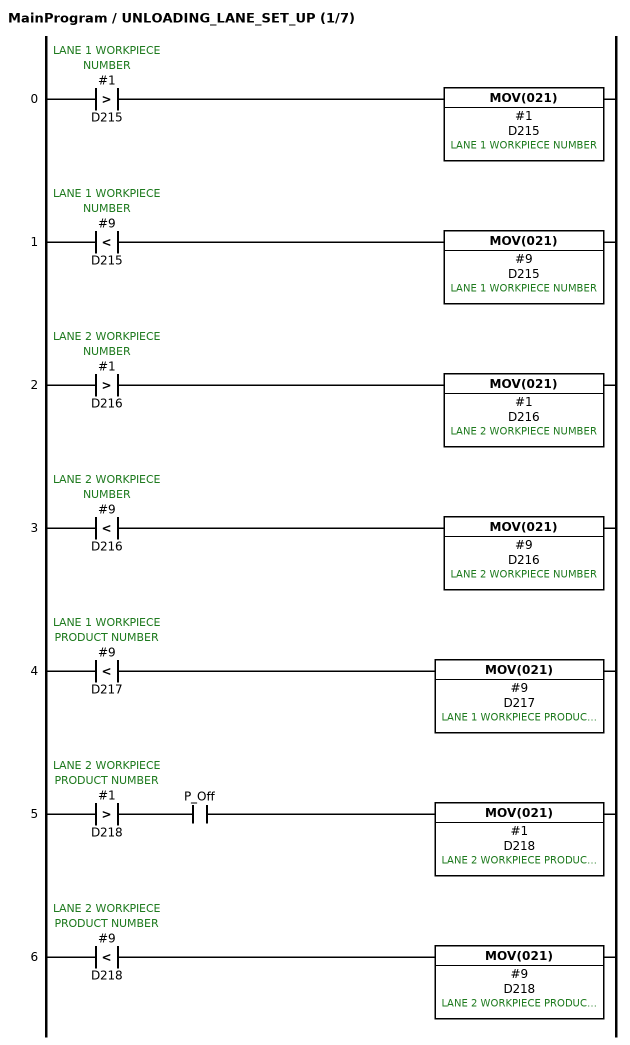
; rung 0
LD>(320) #1 D215  ; LANE 1 WORKPIECE NUMBER
MOV(021) #1 D215  ; LANE 1 WORKPIECE NUMBER
; rung 1
LD<(310) #9 D215  ; LANE 1 WORKPIECE NUMBER
MOV(021) #9 D215  ; LANE 1 WORKPIECE NUMBER
; rung 2
LD>(320) #1 D216  ; LANE 2 WORKPIECE NUMBER
MOV(021) #1 D216  ; LANE 2 WORKPIECE NUMBER
; rung 3
LD<(310) #9 D216  ; LANE 2 WORKPIECE NUMBER
MOV(021) #9 D216  ; LANE 2 WORKPIECE NUMBER
; rung 4
LD<(310) #9 D217  ; LANE 1 WORKPIECE PRODUCT NUMBER
MOV(021) #9 D217  ; LANE 1 WORKPIECE PRODUCT NUMBER
; rung 5
LD>(320) #1 D218  ; LANE 2 WORKPIECE PRODUCT NUMBER
AND P_Off
MOV(021) #1 D218  ; LANE 2 WORKPIECE PRODUCT NUMBER
; rung 6
LD<(310) #9 D218  ; LANE 2 WORKPIECE PRODUCT NUMBER
MOV(021) #9 D218  ; LANE 2 WORKPIECE PRODUCT NUMBER

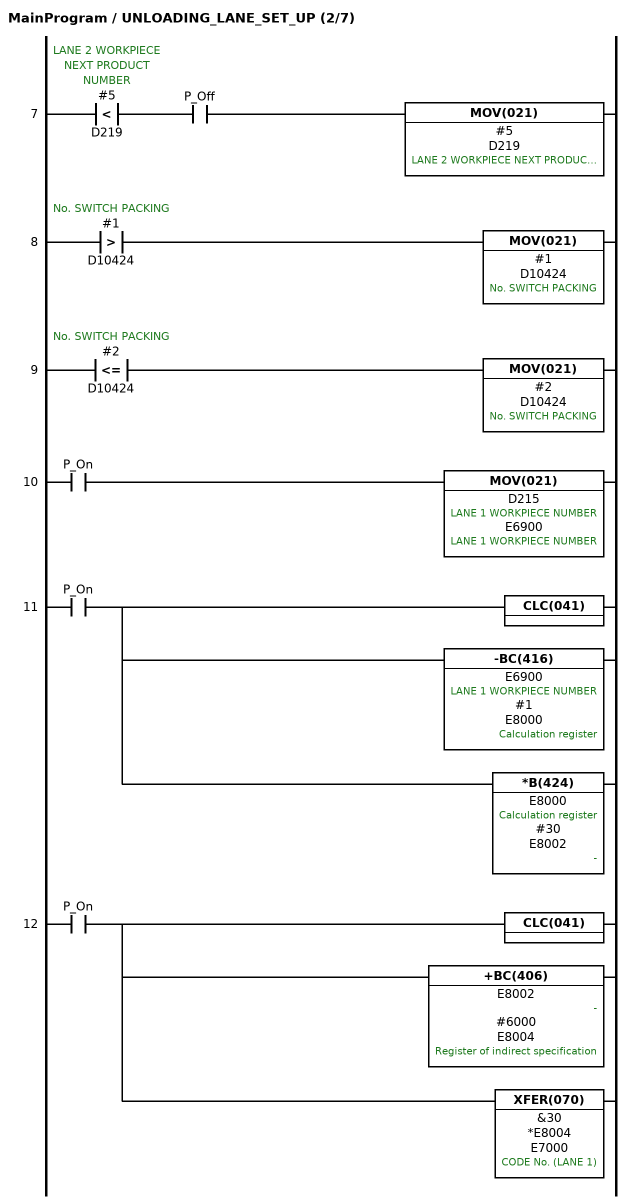
; rung 7
LD<(310) #5 D219  ; LANE 2 WORKPIECE NEXT PRODUCT NUMBER
AND P_Off
MOV(021) #5 D219  ; LANE 2 WORKPIECE NEXT PRODUCT NUMBER
; rung 8
LD>(320) #1 D10424  ; No. SWITCH PACKING
MOV(021) #1 D10424  ; No. SWITCH PACKING
; rung 9
LD<=(315) #2 D10424  ; No. SWITCH PACKING
MOV(021) #2 D10424  ; No. SWITCH PACKING
; rung 10
LD P_On
MOV(021) D215 E6900  ; LANE 1 WORKPIECE NUMBER
; rung 11
LD P_On
CLC(041)
-BC(416) E6900 #1 E8000  ; LANE 1 WORKPIECE NUMBER, Calculation register
*B(424) E8000 #30 E8002  ; Calculation register, -
; rung 12
LD P_On
CLC(041)
+BC(406) E8002 #6000 E8004  ; -, Register of indirect specification
XFER(070) &30 *E8004 E7000  ; CODE No. (LANE 1)

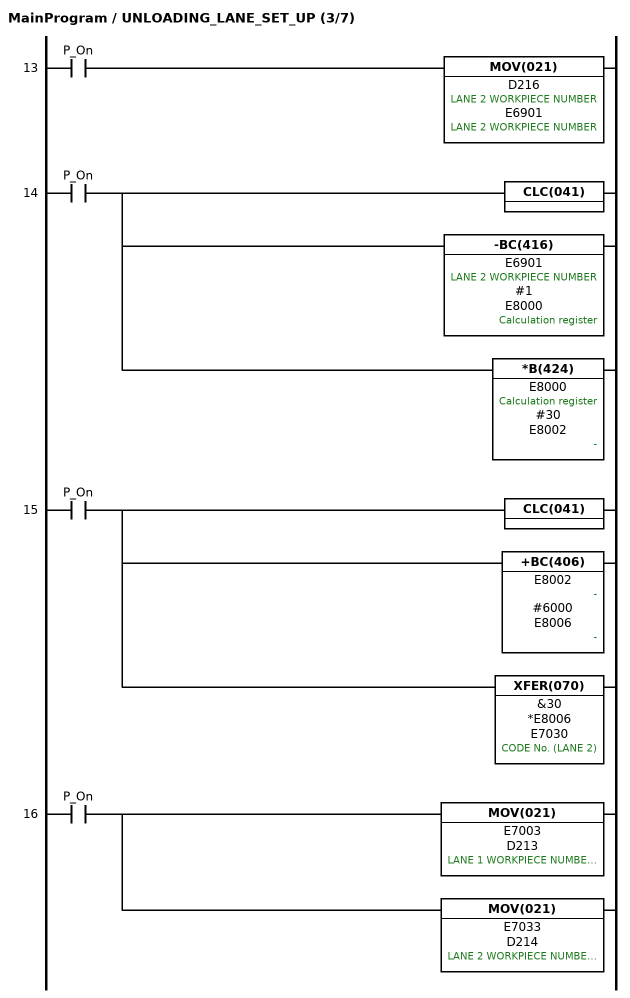
; rung 13
LD P_On
MOV(021) D216 E6901  ; LANE 2 WORKPIECE NUMBER
; rung 14
LD P_On
CLC(041)
-BC(416) E6901 #1 E8000  ; LANE 2 WORKPIECE NUMBER, Calculation register
*B(424) E8000 #30 E8002  ; Calculation register, -
; rung 15
LD P_On
CLC(041)
+BC(406) E8002 #6000 E8006  ; -
XFER(070) &30 *E8006 E7030  ; CODE No. (LANE 2)
; rung 16
LD P_On
MOV(021) E7003 D213  ; LANE 1 WORKPIECE NUMBER DISPLAY
MOV(021) E7033 D214  ; LANE 2 WORKPIECE NUMBER DISPLAY

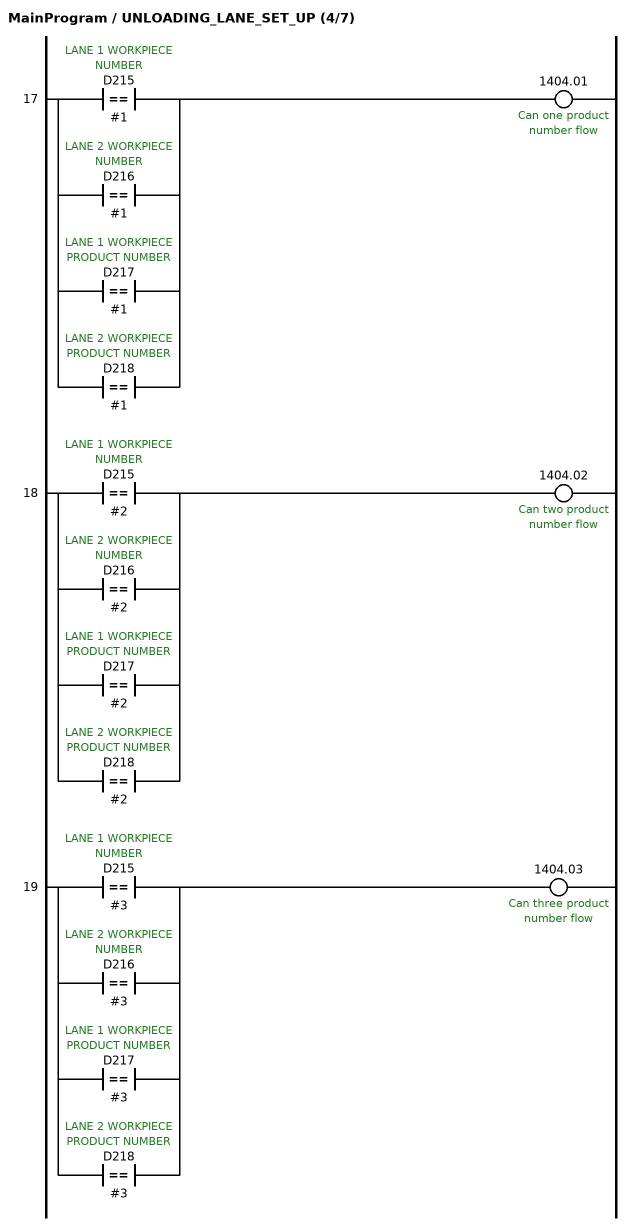
; rung 17
LD=(300) D215 #1  ; LANE 1 WORKPIECE NUMBER
OR=(300) D216 #1  ; LANE 2 WORKPIECE NUMBER
OR=(300) D217 #1  ; LANE 1 WORKPIECE PRODUCT NUMBER
OR=(300) D218 #1  ; LANE 2 WORKPIECE PRODUCT NUMBER
OUT 1404.01  ; Can one product number flow
; rung 18
LD=(300) D215 #2  ; LANE 1 WORKPIECE NUMBER
OR=(300) D216 #2  ; LANE 2 WORKPIECE NUMBER
OR=(300) D217 #2  ; LANE 1 WORKPIECE PRODUCT NUMBER
OR=(300) D218 #2  ; LANE 2 WORKPIECE PRODUCT NUMBER
OUT 1404.02  ; Can two product number flow
; rung 19
LD=(300) D215 #3  ; LANE 1 WORKPIECE NUMBER
OR=(300) D216 #3  ; LANE 2 WORKPIECE NUMBER
OR=(300) D217 #3  ; LANE 1 WORKPIECE PRODUCT NUMBER
OR=(300) D218 #3  ; LANE 2 WORKPIECE PRODUCT NUMBER
OUT 1404.03  ; Can three product number flow

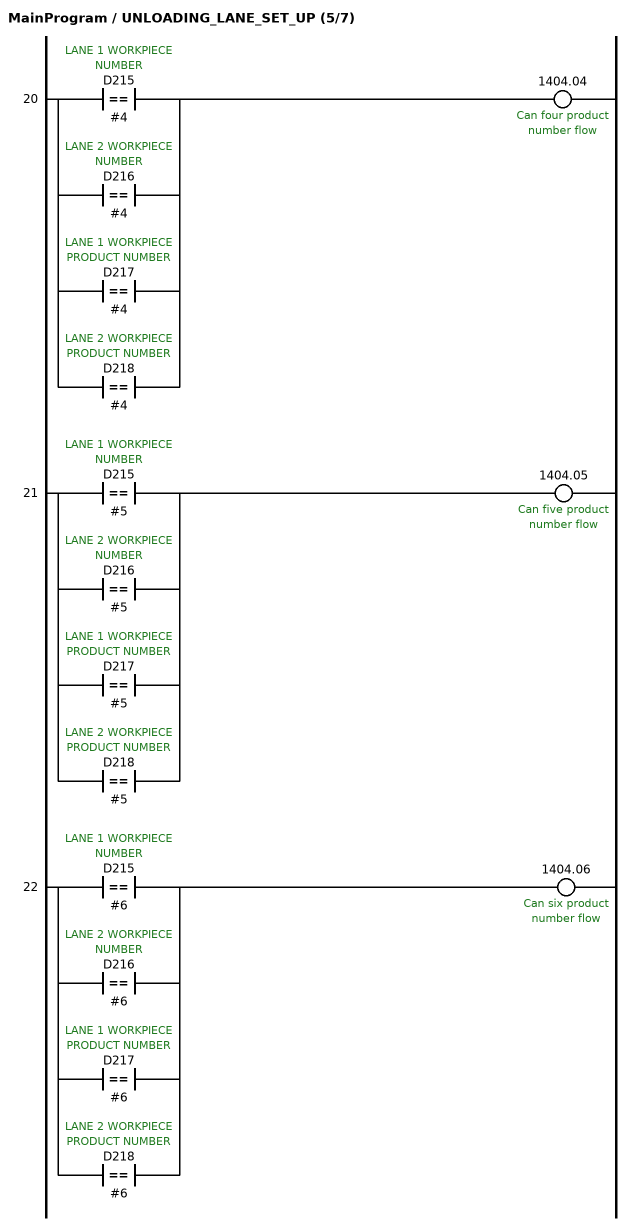
; rung 20
LD=(300) D215 #4  ; LANE 1 WORKPIECE NUMBER
OR=(300) D216 #4  ; LANE 2 WORKPIECE NUMBER
OR=(300) D217 #4  ; LANE 1 WORKPIECE PRODUCT NUMBER
OR=(300) D218 #4  ; LANE 2 WORKPIECE PRODUCT NUMBER
OUT 1404.04  ; Can four product number flow
; rung 21
LD=(300) D215 #5  ; LANE 1 WORKPIECE NUMBER
OR=(300) D216 #5  ; LANE 2 WORKPIECE NUMBER
OR=(300) D217 #5  ; LANE 1 WORKPIECE PRODUCT NUMBER
OR=(300) D218 #5  ; LANE 2 WORKPIECE PRODUCT NUMBER
OUT 1404.05  ; Can five product number flow
; rung 22
LD=(300) D215 #6  ; LANE 1 WORKPIECE NUMBER
OR=(300) D216 #6  ; LANE 2 WORKPIECE NUMBER
OR=(300) D217 #6  ; LANE 1 WORKPIECE PRODUCT NUMBER
OR=(300) D218 #6  ; LANE 2 WORKPIECE PRODUCT NUMBER
OUT 1404.06  ; Can six product number flow

